# EPICS StreamDevice protocol: siteApps-725b29e158e8061764313f5708af9e46fe30c0a8/siteApps-725b29e158e8061764313f5708af9e46fe30c0a8/xgs600/xgs600App/Db/lk224.proto
#
# LakeShore Model 224 Temperature Monitor Stream protocol file
#
# Thursday, July 30 13:58:21 KST 2015, jhlee
#
# - Author  : Jeong Han Lee
# - email   : jhlee@ibs.re.kr
# - license : EPICS open license

Terminator   = CR LF;
ReplyTimeout = 2000;
ReadTimeout  = 1000;

cmd
{
    out "\$1";
}

getIDN
{
    out "*IDN?";
    in  "%s";
    @init {out "*IDN?"; in "%s";}
    ExtraInput = Ignore;
}

getD
{
    out "\$1?";
    in  "%d";
    ExtraInput = Ignore;
}

setD
{
    out "\$1 %d";
    @init { getD; }
}

getLEDS
{
    out "LEDS?";
    in  "%d";
    ExtraInput = Ignore;
}

setLEDS
{
    out "LEDS %{0|1}";
}

getMode
{
    out "MODE?";
    in  "%d";
    ExtraInput = Ignore;
}

setMode
{
    out "MODE %{0|1|2}";
    @init {getMode;}
}

getInName
{
    out "INNAME?";
    in  "%s";
    ExtraInput = Ignore;
}

readCelsius
{
    out "CRDG? \$1";
    in  "%f";
 #   ExtraInput = Ignore;
}

readKelvin
{
    out "KRDG? \$1";
    in  "%f";
#    ExtraInput = Ignore;
}

readSensUnit
{
    out "SRDG? \$1";
    in  "%f";
#    ExtraInput = Ignore;
}

readA_Kelvin
{
    out "KRDG? 0";
    in "%f,%*f,%*f,%*f,%*f,%*f,%*f,%*f,%*f,%*f,%*f,%*f";
    @mismatch {
        in "%s";

    }
}

readB_Kelvin
{
    in "%*f,%f,%*f,%*f,%*f,%*f,%*f,%*f,%*f,%*f,%*f,%*f";
}

readC1_Kelvin
{
    in "%*f,%*f,%f,%*f,%*f,%*f,%*f,%*f,%*f,%*f,%*f,%*f";
}

readC2_Kelvin
{
    in "%*f,%*f,%*f,%f,%*f,%*f,%*f,%*f,%*f,%*f,%*f,%*f";
}

readC3_Kelvin
{
    in "%*f,%*f,%*f,%*f,%f,%*f,%*f,%*f,%*f,%*f,%*f,%*f";
}

readC4_Kelvin
{
    in "%*f,%*f,%*f,%*f,%*f,%f,%*f,%*f,%*f,%*f,%*f,%*f";
}

readC5_Kelvin
{
    in "%*f,%*f,%*f,%*f,%*f,%*f,%f,%*f,%*f,%*f,%*f,%*f";
}

readD1_Kelvin
{
    in "%*f,%*f,%*f,%*f,%*f,%*f,%*f,%f,%*f,%*f,%*f,%*f";
}

readD2_Kelvin
{
    in "%*f,%*f,%*f,%*f,%*f,%*f,%*f,%*f,%f,%*f,%*f,%*f";
}

readD3_Kelvin
{
    in "%*f,%*f,%*f,%*f,%*f,%*f,%*f,%*f,%*f,%f,%*f,%*f";
}

readD4_Kelvin
{
    in "%*f,%*f,%*f,%*f,%*f,%*f,%*f,%*f,%*f,%*f,%f,%*f";
}

readD5_Kelvin
{
    in "%*f,%*f,%*f,%*f,%*f,%*f,%*f,%*f,%*f,%*f,%*f,%f";
}

readRDGST
{
    out "RDGST? \$1";
    in "%d";
}
